DATA_BLOCK "dbArchiveEquipEom"
{ S7_Optimized_Access := 'TRUE' }
VERSION : 0.8
NON_RETAIN
"fbArchiveEquipEom"

BEGIN

END_DATA_BLOCK

